// TwinCAT 3 PLC project AdsStaticNetId
// ProgramVersion: 3.1.4023.0
// libraries:
//   Tc2_DataExchange, * (Beckhoff Automation GmbH)
//   Tc2_Standard, * (Beckhoff Automation GmbH)
//   Tc2_System, * (Beckhoff Automation GmbH)
//   Tc2_Utilities, * (Beckhoff Automation GmbH)
//   Tc3_BA_Common, * (Beckhoff Automation GmbH)
//   Tc3_Module, * (Beckhoff Automation GmbH)
// project tree:
//   DUTs/ AdsData.TcDUT (not stored), AdsSocket.TcPOU (not stored)
//   DUTs/Enums/ AreaNum.TcDUT (not stored), EventsEnum.TcTLEO (not stored)
//   GVLs/ LocalSocket.TcGVL (not stored)
//   / PlcTask.TcTTO (not stored)
//   POUs/ AdsTcp_WinCE.TcPOU (not stored), BufferIsEmpty.TcPOU (not stored), MAIN.TcPOU
// real-time tasks:
//   TASK PlcTask: cycle T#10ms, priority 21, ADS port 350

// ---- POUs/MAIN.TcPOU
PROGRAM MAIN
VAR_OUTPUT
	currentTime : TIMESTRUCT;
END_VAR
VAR
	sMessage : STRING := 'from SERVER to CLIENT';
	newRecipient : STRING;
	newData : AdsData;
	
	sendOnce : BOOL;
	sendFastNum : BOOL;;
	
	retrievedData : AdsData;
	
	i : INT := 0;
	
	fbLocalSystemTime : FB_LocalSystemTime;
	
	messageSize : ULINT;
END_VAR

fbLocalSystemTime(
	sNetID:= , 
	bEnable:= TRUE, 
	dwCycle:= , 
	dwOpt:= , 
	tTimeout:= , 
	bValid=> , 
	systemTime=> currentTime, 
	tzID=> );

AdsTcp_WinCE(
	bBusy=> , 
	err=> , 
	errid=> , 
	areaSockets=> );

IF sendOnce OR sendFastNum THEN
	MEMSET(ADR(newData), 0, SIZEOF(newData));
	
	sMessage := TO_STRING(i);
	
	newRecipient := TO_STRING(AreaNum.AREA_2);
	
	newData.description := EventsEnum.TEST_COMMS;
	newData.timestamp := currentTime;
	MEMCPY(ADR(newData.binaryData), ADR(sMessage), LEN(sMessage));
	
	IF AdsTcp_WinCE.sendMessage(recipient := newRecipient, data := newData) THEN
		i := i + 1;
		sendOnce := FALSE;
	END_IF
	
END_IF

//retrievedData := AdsTcp_WinCE.AREA_2.receivingData;

END_PROGRAM
